Fanuc KAREL source: kx00033.KL

-- PROVISIONAL review KL for V1013-1; original PC SHA256 3aba3b4596d33b43b72c528f991cd967d8f7da7c750021672badbc494f9592f0
-- Incomplete behavior may be omitted. Consult companion uncertainty JSON. Do not deploy.
PROGRAM KX00033
%NOLOCKGROUP
-- UNRESOLVED_DECL I type=fa0010
-- UNRESOLVED_DECL J type=fa0010
-- UNRESOLVED_DECL B type=fa0012
-- UNRESOLVED_DECL F type=fa001d
-- UNRESOLVED_DECL S type=fa1f50
-- UNRESOLVED_DECL P type=fa0102
BEGIN
  -- UNRESOLVED_PC offsets 5-12; opcodes 9D,23
  -- UNRESOLVED_PC offsets 17-21; opcodes 7F
END KX00033
